FUNCTION_BLOCK BATTERYOPTIMIZER_DEB2 (* Optimizes battery charging and/or discharging using PV power and load forecasts with a battery simulation. *)
  (* Standard: 61499-2; Description: IEC 61499 implementation of the "PVprog" algorithm. Original version's MIT license: Copyright (c) 2016 Joseph Bergner, Johannes Weniger, Tjarko Tjaden Permission is hereby granted, free of charge, to any person obtaining a copy of this software and associated documentation files (the "Software"), to deal in the Software without restriction, including without limitation the rights to use, copy, modify, merge, publish, distribute, sublicense, and/or sell copies of the Software, and to permit persons to whom the Software is furnished to do so, subject to the following conditions: The above copyright notice and this permission notice shall be included in all copies or substantial portions of the Software. THE SOFTWARE IS PROVIDED "AS IS", WITHOUT WARRANTY OF ANY KIND, EXPRESS OR IMPLIED, INCLUDING BUT NOT LIMITED TO THE WARRANTIES OF MERCHANTABILITY, FITNESS FOR A PARTICULAR PURPOSE AND NONINFRINGEMENT. IN NO EVENT SHALL THE AUTHORS OR COPYRIGHT HOLDERS BE LIABLE FOR ANY CLAIM, DAMAGES OR OTHER LIABILITY, WHETHER IN AN ACTION OF CONTRACT, TORT OR OTHERWISE, ARISING FROM, OUT OF OR IN CONNECTION WITH THE SOFTWARE OR THE USE OR OTHER DEALINGS IN THE SOFTWARE. *)
  (* Version 1.0, 2017-05-19, Marc Jakobi, HTW Berlin *)
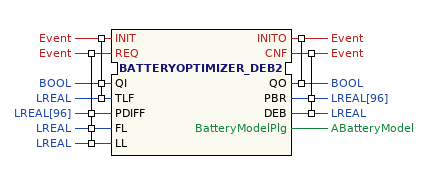
  EVENT_INPUT
    INIT WITH QI, TLF; (* Initialization Request *)
    REQ WITH FL, LL, PDIFF; (* Normal Execution Request *)
  END_EVENT
  EVENT_OUTPUT
    INITO WITH QO; (* Initialization Confirm *)
    CNF WITH PBR, DEB; (* Execution Confirmation *)
  END_EVENT
  VAR_INPUT
    QI : BOOL; (* Input event qualifier *)
    TLF : LREAL := 15; (* Time frame forecasted ahead (looked forward) in h *)
    PDIFF : ARRAY [0..95] OF LREAL; (* Power difference forecast in W (negative = PV deficit, positive = PV surplus) *)
    FL : LREAL; (* Feed-in limitation in W (0 for none) *)
    LL : LREAL; (* Load limit in W (0 for none) *)
  END_VAR
  VAR_OUTPUT
    QO : BOOL; (* Output event qualifier *)
    PBR : ARRAY [0..95] OF LREAL; (* Battery charge/discharge roadmap (Power in W, positive = charge, negative = discharge, 15 min resolved) *)
    DEB : LREAL; (* Debug output *)
  END_VAR
  PLUGS
    BatteryModelPlg : ABatteryModel; (* Link to battery model *)
  END_PLUGS
  VAR
    FLFLAG : BOOL := FALSE; (* True, when feed-in limit optimization is active, false otherwise *)
    LLFLAG : BOOL := FALSE; (* True, when load limit optimization is active, false otherwise *)
    OPTIMIZEDFEEDINLIMIT : LREAL := 0; (* Optimized PV feed-in limitation *)
    OPTIMIZEDLOADLIMIT : LREAL := 0; (* Optimized load limitation *)
    INCFACTOR : LREAL := -1; (* Increment factor for feed-in and load limitation iterators *)
    PCAFTERCHARGE : LREAL := -1; (* Battery capacity after previous charge iteration step *)
    PCAFTERDISCHARGE : LREAL := -1; (* Battery capacity after previous discharge iteration step *)
    FEEDINLIMITITERATOR : LREAL := 0; (* PV feed-in limit iterator for battery simulation *)
    LOADLIMITITERATOR : LREAL := 0; (* Load limit iterator for battery simulation *)
    LOOKFORWARDTIMEINTIMESTEPS : UINT := 60; (* Number of time steps (15 min intervals) to look ahead for forecast *)
  END_VAR
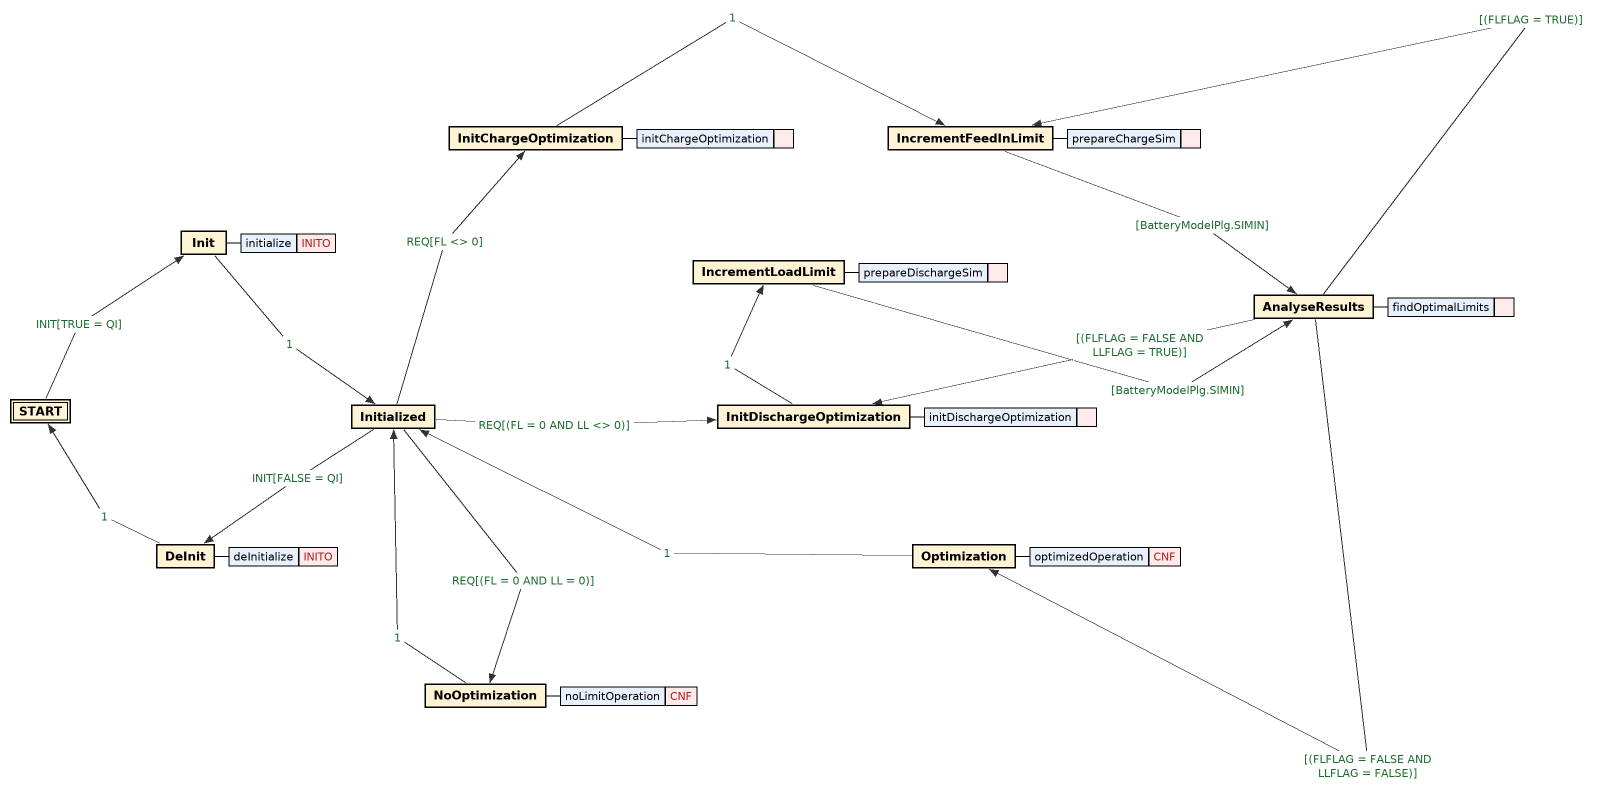
  EC_STATES
    START; (* Initial State *)
    Init : initialize -> INITO; (* Initialization *)
    Initialized;
    DeInit : deInitialize -> INITO;
    IncrementFeedInLimit : prepareChargeSim;
    IncrementLoadLimit : prepareDischargeSim;
    InitChargeOptimization : initChargeOptimization;
    InitDischargeOptimization : initDischargeOptimization;
    NoOptimization : noLimitOperation -> CNF;
    AnalyseResults : findOptimalLimits;
    Optimization : optimizedOperation -> CNF;
  END_STATES
  EC_TRANSITIONS
    START TO Init := INIT[TRUE = QI];
    Init TO Initialized := 1;
    DeInit TO START := 1;
    Initialized TO DeInit := INIT[FALSE = QI];
    Initialized TO InitDischargeOptimization := REQ[(FL = 0 AND LL <> 0)];
    Initialized TO InitChargeOptimization := REQ[FL <> 0];
    Initialized TO NoOptimization := REQ[(FL = 0 AND LL = 0)];
    NoOptimization TO Initialized := 1;
    InitChargeOptimization TO IncrementFeedInLimit := 1;
    InitDischargeOptimization TO IncrementLoadLimit := 1;
    AnalyseResults TO IncrementFeedInLimit := [(FLFLAG = TRUE)];
    AnalyseResults TO InitDischargeOptimization := [(FLFLAG = FALSE AND LLFLAG = TRUE)];
    AnalyseResults TO Optimization := [(FLFLAG = FALSE AND LLFLAG = FALSE)];
    Optimization TO Initialized := 1;
    IncrementFeedInLimit TO AnalyseResults := [BatteryModelPlg.SIMIN];
    IncrementLoadLimit TO AnalyseResults := [BatteryModelPlg.SIMIN];
  END_TRANSITIONS
  ALGORITHM initialize IN ST: (* Initialization algorithm *)
VAR
	tmp1 : LREAL;
	tmp2 : UINT;
END_VAR;
/*
 * Used internal vars & inputs:
 * TLF, LOOKFORWARDTIMEINTIMESTEPS : UINT;
 */
tmp1 := TLF * 4; // output resolution = 15 min
tmp2 := LREAL_TO_UINT(tmp1);
IF UINT_TO_LREAL(tmp2) < tmp1 THEN
 	LOOKFORWARDTIMEINTIMESTEPS := tmp2 + 1;
ELSE
	LOOKFORWARDTIMEINTIMESTEPS := tmp2;
END_IF;
// Set output event qualifier
QO := QI;
  END_ALGORITHM
  ALGORITHM deInitialize IN ST: (* Normally executed algorithm *)
VAR
	i : UINT;
END_VAR;
FOR i := 0 TO 95 BY 1 DO
	PBR[i] := 0;
END_FOR;
QO := FALSE;
  END_ALGORITHM
  ALGORITHM initChargeOptimization IN ST: (* Initializes the PV feed-in limit iteration *)
/*
 * Used internal vars & inputs:
 * INCFACTOR, PCAFTERCHARGE, FL, OPTIMIZEDFEEDINLIMIT : LREAL;
 */
INCFACTOR := -1;
PCAFTERCHARGE := -1;
OPTIMIZEDFEEDINLIMIT := 0;
IF FL < 0 THEN // Make sure feed-in limit is positive
	FL := FL * (-1);
END_IF;
FLFLAG := TRUE;
IF LL = 0 THEN
	LLFLAG := FALSE;
ELSE
	LLFLAG := TRUE;
END_IF;
  END_ALGORITHM
  ALGORITHM noLimitOperation IN ST: (* Calculates the battery charge roadmap without feed-in and load limits *)
VAR
	i : UINT;
END_VAR;
/*
 * Used internal vars & inputs:
 * PDIFF, PBR : LREAL;
 * LOOKFORWARDTIMEINTIMESTEPS : UINT;
 */
 FOR i := 0 TO LOOKFORWARDTIMEINTIMESTEPS BY 1 DO
 	PBR[i] := PDIFF[i];
 END_FOR;
  END_ALGORITHM
  ALGORITHM prepareChargeSim IN ST: (* Prepares the data for the battery charging simulation *)
VAR
	i : UINT;
    pvSurplus : LREAL;
END_VAR;
/*
 * Used internal vars & inputs:
 * INCFACTOR, FEEDINLIMITITERATOR, FL, PM, TLF : LREAL;
 * LOOKFORWARDTIMEINTIMESTEPS : UINT;
 */
// Increment feed-in limit iterator
INCFACTOR := INCFACTOR + 1;
FEEDINLIMITITERATOR := INCFACTOR * FL / 100;
BatteryModelPlg.ECD := 0; // Initialize mean battery charging power
FOR i := 0 TO LOOKFORWARDTIMEINTIMESTEPS - 1 BY 1 DO
	// Increment with PV surpluses above feed-in limit iterator
	pvSurplus := PDIFF[i] - FEEDINLIMITITERATOR;
	IF pvSurplus < 0 THEN
		pvSurplus := 0;
	END_IF;
	BatteryModelPlg.ECD := BatteryModelPlg.ECD + pvSurplus;
END_FOR;
// Calculate charging energy over forecast horizon in kWh
BatteryModelPlg.ECD := (BatteryModelPlg.ECD / UINT_TO_LREAL(LOOKFORWARDTIMEINTIMESTEPS)) / 1000 * TLF ;
  END_ALGORITHM
  ALGORITHM findOptimalLimits IN ST: (* Analyses the battery charge/discharge simulation results *)
/*
 * Used internal vars & inputs:
 * FEEDINLIMITITERATOR, LOADLIMITITERATOR, FL, LL, CSIM : LREAL;
 * PCAFTERCHARGE, OPTIMIZEDFEEDINLIMIT, PCAFTERDISCHARGE, OPTIMIZEDLOADLIMIT : LREAL;
 * FLFLAG, LLFLAG : BOOL;
 */
IF FLFLAG THEN
	// Make sure feed-in limit iteration does not go past set limit
	// and find highest possible feed-in limit with maximum possible charge
	// capacity to cover limitation with battery, i.e. stop incrementing feed-in
	// limitation if resulting battery capacity after charge is reduced.
	IF (BatteryModelPlg.CSIM < PCAFTERCHARGE OR FEEDINLIMITITERATOR > FL) THEN
		FLFLAG := FALSE;
	ELSE
		OPTIMIZEDFEEDINLIMIT := FEEDINLIMITITERATOR;
		PCAFTERCHARGE := BatteryModelPlg.CSIM;
	END_IF;
ELSE
	// Make sure load limit iteration does not go past set limit
	// and find highest possible load limitation while emptying the battery
	// as much as possible to cover the peak load, i.e. stop incrementing
	// load limit if resulting battery capacity after discharge is increased.
	// PCAFTERDISCHARGE is -1 in initial step.
	IF (PCAFTERDISCHARGE > 0 AND (BatteryModelPlg.CSIM > PCAFTERDISCHARGE OR LOADLIMITITERATOR > LL)) THEN
		LLFLAG := FALSE;
	ELSE
		OPTIMIZEDLOADLIMIT := LOADLIMITITERATOR;
		PCAFTERDISCHARGE := BatteryModelPlg.CSIM;
	END_IF;
END_IF;
IF OPTIMIZEDLOADLIMIT > 0 THEN
	DEB := OPTIMIZEDLOADLIMIT;
END_IF;
  END_ALGORITHM
  ALGORITHM prepareDischargeSim IN ST: (* Prepares the data for the battery discharging simulation *)
VAR
	i : UINT;
    loadDeficit : LREAL;
END_VAR;
/*
 * Used internal vars & inputs:
 * INCFACTOR, LOADLIMITITERATOR, LL, PM : LREAL;
 * LOOKFORWARDTIMEINTIMESTEPS : UINT;
 */
// Increment feed-in limit iterator
INCFACTOR := INCFACTOR + 1;
LOADLIMITITERATOR := INCFACTOR * LL / 100;
BatteryModelPlg.ECD := 0; // Initialize mean battery discharging power
FOR i := 0 TO LOOKFORWARDTIMEINTIMESTEPS - 1 BY 1 DO
	// Increment with PV surpluses above feed-in limit iterator
	loadDeficit := PDIFF[i];
	// workaround for MAX(0, ABS(MIN(0, PFIFF[i])) - LOADLIMITITERATOR)
	IF loadDeficit > 0 THEN
		loadDeficit := 0;
	ELSE
		loadDeficit := loadDeficit * (-1) - LOADLIMITITERATOR;
		IF loadDeficit < 0 THEN
			loadDeficit := 0;
		END_IF;
	END_IF;
	BatteryModelPlg.ECD := BatteryModelPlg.ECD + loadDeficit;
END_FOR;
// Calculate discharging energy over forecast horizon in kWh (negative to indicate discharging)
BatteryModelPlg.ECD := BatteryModelPlg.ECD / UINT_TO_LREAL(LOOKFORWARDTIMEINTIMESTEPS) / 1000 * TLF * (-1);
  END_ALGORITHM
  ALGORITHM initDischargeOptimization IN ST: (* Initializes the load limit iteration *)
/*
 * Used internal vars & inputs:
 * INCFACTOR, PCAFTERDISCHARGE, OPTIMIZEDLOADLIMIT, LL : LREAL;
 */
INCFACTOR := -1;
PCAFTERDISCHARGE := -1;
OPTIMIZEDLOADLIMIT := 0;
IF LL < 0 THEN // Make sure load limit is positive
	LL := LL * (-1);
END_IF;
// Set FLFLAG false to prevent PV feed-in limitation iteration
FLFLAG := FALSE;
LLFLAG := TRUE;
  END_ALGORITHM
  ALGORITHM optimizedOperation IN ST: (* Calculates the battery charge roadmap with optimized feed-in and load limits *)
VAR
	i : UINT;
	batteryChargeForecast : LREAL;
END_VAR;
/*
 * Used internal vars & inputs:
 * FL, LL, PDIFF, PBR, OPTIMIZEDFEEDINLIMIT, OPTIMIZEDLOADLIMIT : LREAL;
 * LOOKFORWARDTIMEINTIMESTEPS : UINT;
 */
IF (FL > 0 AND LL = 0) THEN // Only PV feed-in limitation
	FOR i := 0 TO LOOKFORWARDTIMEINTIMESTEPS - 1 BY 1 DO
		batteryChargeForecast := PDIFF[i] - OPTIMIZEDFEEDINLIMIT;
		IF batteryChargeForecast < 0 THEN // Only look at PV surpluses
			batteryChargeForecast := 0;
		END_IF;
		IF batteryChargeForecast < PDIFF[i] THEN
			PBR[i] := INT_TO_LREAL(LREAL_TO_INT(batteryChargeForecast)); // ROUND() workaround
		ELSE
			PBR[i] := INT_TO_LREAL(LREAL_TO_INT(PDIFF[i]));
		END_IF;
	END_FOR;
ELSIF (FL = 0 AND LL <> 0) THEN // Only load peak shaving
	FOR i := 0 TO LOOKFORWARDTIMEINTIMESTEPS - 1 BY 1 DO
		batteryChargeForecast := PDIFF[i] + OPTIMIZEDLOADLIMIT;
		IF batteryChargeForecast > 0 THEN // Only look at load deficits
			batteryChargeForecast := 0;
		END_IF;
		IF batteryChargeForecast > PDIFF[i] THEN
			PBR[i] := INT_TO_LREAL(LREAL_TO_INT(batteryChargeForecast));
		ELSE
			PBR[i] := INT_TO_LREAL(LREAL_TO_INT(PDIFF[i]));
		END_IF;
	END_FOR;
ELSIF (FL <> 0 AND LL <> 0) THEN // Both PV feed-in limitation and load peak shaving
	FOR i := 0 TO LOOKFORWARDTIMEINTIMESTEPS - 1 BY 1 DO
		IF PDIFF[i] > 0 THEN // PV surplus
			batteryChargeForecast := PDIFF[i] - OPTIMIZEDFEEDINLIMIT;
			IF batteryChargeForecast > 0 THEN
				batteryChargeForecast := 0;
			END_IF;
			IF batteryChargeForecast > PDIFF[i] THEN
				PBR[i] :=INT_TO_LREAL(LREAL_TO_INT(batteryChargeForecast));
			ELSE
				PBR[i] := INT_TO_LREAL(LREAL_TO_INT(PDIFF[i]));
			END_IF;
		ELSE // Load deficit
			batteryChargeForecast := PDIFF[i] + OPTIMIZEDLOADLIMIT;
			IF batteryChargeForecast > 0 THEN
				batteryChargeForecast := 0;
			END_IF;
			IF batteryChargeForecast > PDIFF[i] THEN
				PBR[i] := INT_TO_LREAL(LREAL_TO_INT(batteryChargeForecast));
			ELSE
				PBR[i] := INT_TO_LREAL(LREAL_TO_INT(PDIFF[i]));
			END_IF;
		END_IF;
	END_FOR;
END_IF;
  END_ALGORITHM
END_FUNCTION_BLOCK
